(* IEC 61131-3 sources: horner-cscape-mcp/artifacts/projects/C6_Native_Run/pous, 2 files *)

(* ---- ScaleAnalogFilter.st ---- *)
FUNCTION_BLOCK ScaleAnalogFilter
VAR_INPUT
    RawInput : REAL;
    SmoothingFactor : REAL;
    LowLimit : REAL;
    HighLimit : REAL;
END_VAR
VAR_OUTPUT
    FilteredVal : REAL;
    AlarmHigh : BOOL;
END_VAR
VAR
    ClampedInput : REAL;
END_VAR

(* Clamping raw input to engineering unit limits *)
IF RawInput < LowLimit THEN
    ClampedInput := LowLimit;
ELSIF RawInput > HighLimit THEN
    ClampedInput := HighLimit;
ELSE
    ClampedInput := RawInput;
END_IF;

(* First-order exponential smoothing filter *)
FilteredVal := (SmoothingFactor * ClampedInput) + ((1.0 - SmoothingFactor) * FilteredVal);

(* High alarm threshold at 95% high range *)
IF FilteredVal >= (HighLimit * 0.95) THEN
    AlarmHigh := TRUE;
ELSE
    AlarmHigh := FALSE;
END_IF;

END_FUNCTION_BLOCK

(* ---- MainProcessControl.st ---- *)
PROGRAM MainProcessControl
VAR
    RawSensor1 : REAL := 45.0;
    RawSensor2 : REAL := 78.5;
    Alpha : REAL := 0.25;
    MinRange : REAL := 0.0;
    MaxRange : REAL := 100.0;

    Filter1 : ScaleAnalogFilter;
    Filter2 : ScaleAnalogFilter;

    OutFiltered1 : REAL := 0.0;
    OutFiltered2 : REAL := 0.0;
    Alarm1 : BOOL := FALSE;
    Alarm2 : BOOL := FALSE;
END_VAR

(* C6_MCP_ROUNDTRIP: Native Rung 1 Primary Sensor Filter Active - Verified at 2026-09-08 15:21:23 via FastMCP *)
Filter1(RawInput := RawSensor1, SmoothingFactor := Alpha, LowLimit := MinRange, HighLimit := MaxRange);
OutFiltered1 := Filter1.FilteredVal;
Alarm1 := Filter1.AlarmHigh;

(* Invoke Instance 2: Secondary Redundant Sensor *)
Filter2(RawInput := RawSensor2, SmoothingFactor := Alpha, LowLimit := MinRange, HighLimit := MaxRange);
OutFiltered2 := Filter2.FilteredVal;
Alarm2 := Filter2.AlarmHigh;

END_PROGRAM
